FUNCTION_BLOCK FB_StationT3
VAR_IN_OUT
	XpMover			: MC_PlanarMover;
	XpTrack			: ARRAY [*] OF MC_PlanarTrack;
END_VAR
VAR_INPUT
	execute			: BOOL;
END_VAR
VAR_OUTPUT
	bOccupied		: BOOL;
	bBeforeRotate	: BOOL;
	bReady			: BOOL;
	bDone			: BOOL;
END_VAR
VAR
	nState			: INT;
	fbMoveTrack		: FB_XpMoveTrack;
	fbMoveC			: FB_XpMoveC;
	nTargetTrack	: INT;
	bMove			: BOOL;
	bMoveC			: BOOL;
	nRotatePos		: LREAL :=0;
END_VAR

CASE nState OF
	0: //init
	IF execute THEN
		bOccupied := TRUE;//Stationの状態をOccupiedにする
		bReady := FALSE;
		nState := 20;
	END_IF	
	
	20://移動
	bMove:= TRUE;
	bDone	:= FALSE;
	nTargetTrack:= E_TrackName.T3_2_ToRotate;
	fbMoveTrack.execute := TRUE;

	IF fbMoveTrack.done THEN
		fbMoveTrack.execute:= FALSE;
		bOccupied := FALSE;
		bReady := TRUE;//Stationの状態をReadyにする
		bBeforeRotate := TRUE;//Rotate前の位置まで移動したことをT2に伝える
		bMove:= FALSE;
		nState := 30;
	END_IF
	
	30://回転
	bMoveC := TRUE;
	fbMoveC.execute:= TRUE;
	
	IF fbMoveC.done THEN
		fbMoveC.execute := FALSE;
		bBeforeRotate := FALSE;
		bMoveC:= FALSE;
		nState := 40;
	END_IF
	
	40://T1まで移動
	nTargetTrack:= E_TrackName.T1_1_ToRotate;
	fbMoveTrack.execute:= TRUE;
	bOccupied := FALSE;
	nState := 50;
	
	50:
	IF fbMoveTrack.done THEN
		fbMoveTrack.execute := FALSE;//移動指令を落とす
		bReady :=TRUE;
		bDone :=TRUE;
		nState := 100;
	END_IF

	100://initへ戻る
	nState := 0;
END_CASE

//IF bMove THEN
	fbMoveTrack(XpMover:= XpMover, 
				XpTrack:= XpTrack[nTargetTrack]);
//ELSIF bMoveC THEN	
	fbMoveC(XpMover:= XpMover, 
			position:= nRotatePos + 360);
//END_IF

END_FUNCTION_BLOCK

(* stored: Version 1.1.0.1
   POU FB_StationT3: Id {3370e601-15df-494f-b398-5d30079df286}, SpecialFunc None *)
